// TIA Portal project "P5" (V17)

(* hardware
DEVICE "S7-1500/ET200MP station_1"  S7-1500 station
   slot 0: "Rail_0"  Rack  6ES7 590-1***0-0AA0
   slot 1: "PLC_1"  CPU 1515-2 PN  6ES7 515-2AM02-0AB0  V2.9
      slot 3: "CPU display_1"  6ES7591-1BA00-0AA0
      slot 32768: "PROFINET interface_1"  X1
         slot 32769: "Port_1"  X1 P1
         slot 32770: "Port_2"  X1 P2
      slot 33024: "PROFINET interface_2"  X2
         slot 33025: "Port_1"  X2 P1
      slot 34817: "Virtual CP interface port_1"  Virtual CP interface port  Virtual CP interface port
*)

// ===== PLC "PLC_1"  CPU 1515-2 PN =====

VAR_GLOBAL   // PLC tag table "Default tag table"
   "START" AT %E0.0 : Bool;
   "STOP" AT %E0.1 : Bool;
   "LOAD CELL 1" AT %E0.2 : Bool;
   "LOAD CELL 2" AT %E0.3 : Bool;
   "CYCLE ON" AT %A0.0 : Bool;
   "CONVEYOR  1 MOTOR" AT %A0.1 : Bool;
   "CONVEYOR 2 MOTOR" AT %A0.2 : Bool;
   "FEEDER MOTOR" AT %A0.3 : Bool;
END_VAR

ORGANIZATION_BLOCK "Main"   // OB1, LAD, ProgramCycle
TITLE = "Main Program Sweep (Cycle)"
{ S7_Optimized_Access := 'TRUE' }
VERSION : 0.1
   VAR_INPUT
      Initial_Call : Bool;   // Initial call of this OB
      Remanence : Bool;   // =True, if remanent data are available
   END_VAR
BEGIN

REGION Network 1
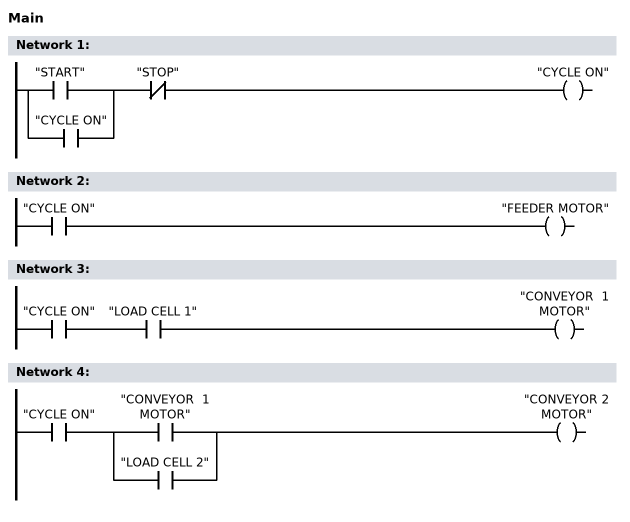
   RUNG wire#powerrail
      Contact( "START" )
      wire#w1
      I_Contact( "STOP" )
      Coil( "CYCLE ON" )
   END_RUNG
   RUNG wire#powerrail
      Contact( "CYCLE ON" )
   END_RUNG wire#w1
   // the same network as SCL:
   "CYCLE ON" := ("START" OR "CYCLE ON") AND NOT "STOP";
END_REGION

REGION Network 2
   RUNG wire#powerrail
      Contact( "CYCLE ON" )
      Coil( "FEEDER MOTOR" )
   END_RUNG
   // the same network as SCL:
   "FEEDER MOTOR" := "CYCLE ON";
END_REGION

REGION Network 3
   RUNG wire#powerrail
      Contact( "CYCLE ON" )
      Contact( "LOAD CELL 1" )
      Coil( "CONVEYOR  1 MOTOR" )
   END_RUNG
   // the same network as SCL:
   "CONVEYOR  1 MOTOR" := "CYCLE ON" AND "LOAD CELL 1";
END_REGION

REGION Network 4
   RUNG wire#powerrail
      Contact( "CYCLE ON" )
      wire#w1
      Contact( "CONVEYOR  1 MOTOR" )
      wire#w2
      Coil( "CONVEYOR 2 MOTOR" )
   END_RUNG
   RUNG wire#w1
      Contact( "LOAD CELL 2" )
   END_RUNG wire#w2
   // the same network as SCL:
   "CONVEYOR 2 MOTOR" := "CYCLE ON" AND ("CONVEYOR  1 MOTOR" OR "LOAD CELL 2");
END_REGION
END_ORGANIZATION_BLOCK